PROGRAM P_Demo_FB_DMXGetDMX512StartAddress
VAR
    fbGetStartAddr    : FB_DMXGetDMX512StartAddress;  // 读起始地址
    stDmxCmdBuffer    : ST_DMXCommandBuffer;          // 与通讯 FB 共用
    wTargetManufId    : WORD := 16#4241;              // 目标灯具厂商 ID
    dwTargetDeviceId  : DWORD := 16#12131415;         // 目标灯具设备 ID
    byTargetPort      : BYTE := 0;                    // 根设备通道 0
    bDoRead           : BOOL := FALSE;                // 在线给一次上升沿触发
    bBusy             : BOOL;
    bError            : BOOL;
    udiErrId          : UDINT;
    iStartAddr        : INT;                          // DMX512 起始地址(1-512;0xFFFF=不占槽)
END_VAR

// ============================================================
// Tc2_DMX.FB_DMXGetDMX512StartAddress 演示程序
// ============================================================
// 场景：地址规划核对：上电后批量读出每盏灯 DMX512 起始地址，与设计图纸比对，发现冲突及时纠正。
// 价值：把现场实际起始地址读进 PLC 与设计值自动比对，避免因地址冲突导致多盏灯同动作。
// 验证：给 bDoRead 一次上升沿 -> bBusy 短暂 TRUE -> 回 FALSE 后 iStartAddr 即设备起始地址(1-512)；纯 RDM 不占槽设备返回 0xFFFF(=-1 按 INT 显示或 65535)。
// 验证步骤：
//   1. 右键 PLC 项目下 POUs 文件夹 → Add → Existing Item → 选本 .TcPOU 文件
//   2. 引用 Tc2_DMX；同项目里放一个 FB_EL6851CommunicationEx 实例并共用 stDmxCmdBuffer（非 CycleMode）
//   3. 编译 → 登录 → 运行；按上方『验证』行在线给上升沿观察
// ============================================================

fbGetStartAddr(
    bStart                     := bDoRead,
    wDestinationManufacturerId := wTargetManufId,
    dwDestinationDeviceId      := dwTargetDeviceId,
    byPortId                   := byTargetPort,
    dwOptions                  := 0,
    stCommandBuffer            := stDmxCmdBuffer,
    bBusy                      => bBusy,
    bError                     => bError,
    udiErrorId                 => udiErrId,
    iDMX512StartAddress        => iStartAddr
);

END_PROGRAM

(* stored: Version 1.1.0.1, ProductVersion 3.1.4024.5
   POU P_Demo_FB_DMXGetDMX512StartAddress: Id {145e0f5b-3159-5366-81f0-cb95592e9af2}, SpecialFunc None *)
